// TIA Portal V18 export
TYPE "MEStoPLC_Common_ext"
// stored: IsFailsafeCompliant false
   STRUCT
      "M-HeartBeat" : Bool;   // MES心跳信号，频率5S，PLC10S延迟判定报警
   END_STRUCT;
END_TYPE
